FUNCTION_BLOCK FB_EmergencyStop
VAR_INPUT
END_VAR
VAR_OUTPUT
END_VAR
VAR
END_VAR

CASE emergencySubState OF

	step0:	//setting of OPCUA variables
			Module2101.Output.SkillOutput.SkillOutput0.Busy := FALSE;
			Module2101.Output.SkillOutput.SkillOutput0.Done := FALSE;
			Module2101.Output.SkillOutput.SkillOutput0.Dummy := FALSE;
			Module2101.Output.SkillOutput.SkillOutput0.Error := TRUE;
			Module2101.Output.SkillOutput.SkillOutput0.Ready := FALSE;
			//go into the right error state
			Module2101.Output.ErrorID := 2;
			Module2101.Output.CurrentTaskDescription := 'Emergency stop';
			Module2101.Output.Error := TRUE;
			Module2101.Output.ErrorDescription := 'Emergency stop';
			
			//wait for process tool to set the module in manual mode
			IF(Module2101.Input.Mode = DUT_MODE.Manual) THEN
				emergencySubState := step1;
			END_IF
			
	step1:	//wait for process tool to set the module in init mode
			IF(Module2101.Input.Mode = DUT_MODE.Auto) THEN
				//reset error 
				Module2101.Output.Error := FALSE;
				Module2101.Output.ErrorDescription := '';
				Module2101.Output.ErrorID := 0;
				
				//change to init state
				initSubState := step0;
				mainState := eMainState.init;
				emergencySubState := step0;
			END_IF
			
			
	step2:	
			
	step3:	

END_CASE

END_FUNCTION_BLOCK

(* stored: Version 1.1.0.1, ProductVersion 3.1.0.25
   POU FB_EmergencyStop: Id {2676421f-a439-4c78-876b-2d65f5154178} *)
